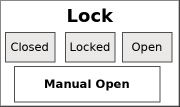
VISUALIZATION vLockFrame  // 180x107
VAR_INPUT
	iNameIndex :INT;
END_VAR
VAR_IN_OUT
	fbLock :FB_Lock;

END_VAR
    Rectangle (0,0 180x107)
    Rectangle (5,32 50x30), "Closed", colour toggle: fbLock.prClosed
    Rectangle (39,1 102x30), "Lock", text list: 'tlDevices', text index: iNameIndex
    Rectangle (65,32 50x30), "Locked", colour toggle: fbLock.prClosedAndLocked
    Rectangle (122,32 50x30), "Open", colour toggle: fbLock.stInOut.bOpen
    Rectangle (14,66 146x36), "Manual Open", input disabled if: NOT fbLock.bReleaseManulOpening
        OnMouseDown: execute { fbLock.mManualOpen(); }
END_VISUALIZATION

(* stored: Version 1.1.0.1, ProductVersion 3.1.4024.15
   Visu vLockFrame: Id {dd2aa803-bd21-4f31-a982-a3a97863a71c} *)
